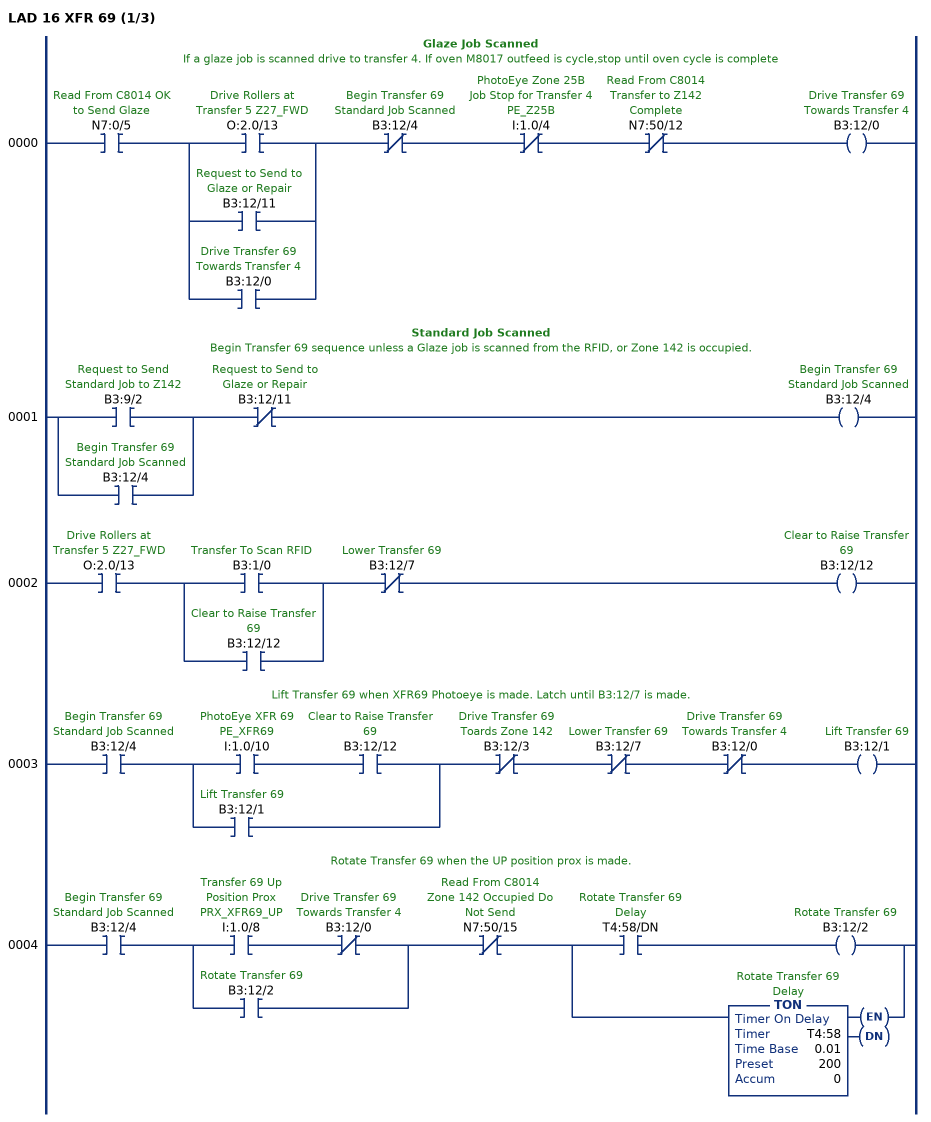
% Rung: 0 %
% TITLE: Glaze Job Scanned %
% If a glaze job is scanned drive to transfer 4. If oven M8017 outfeed is cycle,stop until oven cycle is complete %
SOR XIC N7:0/5 BST XIC O:2.0/13 NXB XIC B3:12/11 NXB XIC B3:12/0 BND XIO B3:12/4 XIO I:1.0/4 XIO N7:50/12 OTE B3:12/0 EOR
%   N7:0/5  "Read From C8014 OK to Send Glaze" %
%   O:2.0/13  Z27_FWD  "Drive Rollers at Transfer 5" %
%   B3:12/11  "Request to Send to Glaze or Repair" %
%   B3:12/0  "Drive Transfer 69 Towards Transfer 4" %
%   B3:12/4  "Begin Transfer 69 Standard Job Scanned" %
%   I:1.0/4  PE_Z25B  "PhotoEye Zone 25B Job Stop for Transfer 4" %
%   N7:50/12  "Read From C8014 Transfer to Z142 Complete" %
% Rung: 1 %
% TITLE: Standard Job Scanned %
% Begin Transfer 69 sequence unless a Glaze job is scanned from the RFID, or Zone 142 is occupied. %
SOR BST XIC B3:9/2 NXB XIC B3:12/4 BND XIO B3:12/11 OTE B3:12/4 EOR
%   B3:9/2  "Request to Send Standard Job to Z142" %
%   B3:12/4  "Begin Transfer 69 Standard Job Scanned" %
%   B3:12/11  "Request to Send to Glaze or Repair" %
% Rung: 2 %
SOR XIC O:2.0/13 BST XIC B3:1/0 NXB XIC B3:12/12 BND XIO B3:12/7 OTE B3:12/12 EOR
%   O:2.0/13  Z27_FWD  "Drive Rollers at Transfer 5" %
%   B3:1/0  "Transfer To Scan RFID" %
%   B3:12/12  "Clear to Raise Transfer 69" %
%   B3:12/7  "Lower Transfer 69" %
% Rung: 3 %
% Lift Transfer 69 when XFR69 Photoeye is made. Latch until B3:12/7 is made. %
SOR XIC B3:12/4 BST XIC I:1.0/10 XIC B3:12/12 NXB XIC B3:12/1 BND XIO B3:12/3 XIO B3:12/7 XIO B3:12/0 OTE B3:12/1 EOR
%   B3:12/4  "Begin Transfer 69 Standard Job Scanned" %
%   I:1.0/10  PE_XFR69  "PhotoEye XFR 69" %
%   B3:12/12  "Clear to Raise Transfer 69" %
%   B3:12/1  "Lift Transfer 69" %
%   B3:12/3  "Drive Transfer 69 Toards Zone 142" %
%   B3:12/7  "Lower Transfer 69" %
%   B3:12/0  "Drive Transfer 69 Towards Transfer 4" %
% Rung: 4 %
% Rotate Transfer 69 when the UP position prox is made. %
SOR XIC B3:12/4 BST XIC I:1.0/8 XIO B3:12/0 NXB XIC B3:12/2 BND XIO N7:50/15 BST XIC T4:58/DN OTE B3:12/2 NXB TON T4:58 0.01 200 0 BND EOR
%   B3:12/4  "Begin Transfer 69 Standard Job Scanned" %
%   I:1.0/8  PRX_XFR69_UP  "Transfer 69 Up Position Prox" %
%   B3:12/0  "Drive Transfer 69 Towards Transfer 4" %
%   B3:12/2  "Rotate Transfer 69" %
%   N7:50/15  "Read From C8014 Zone 142 Occupied Do Not Send" %
%   T4:58  "Rotate Transfer 69 Delay" %

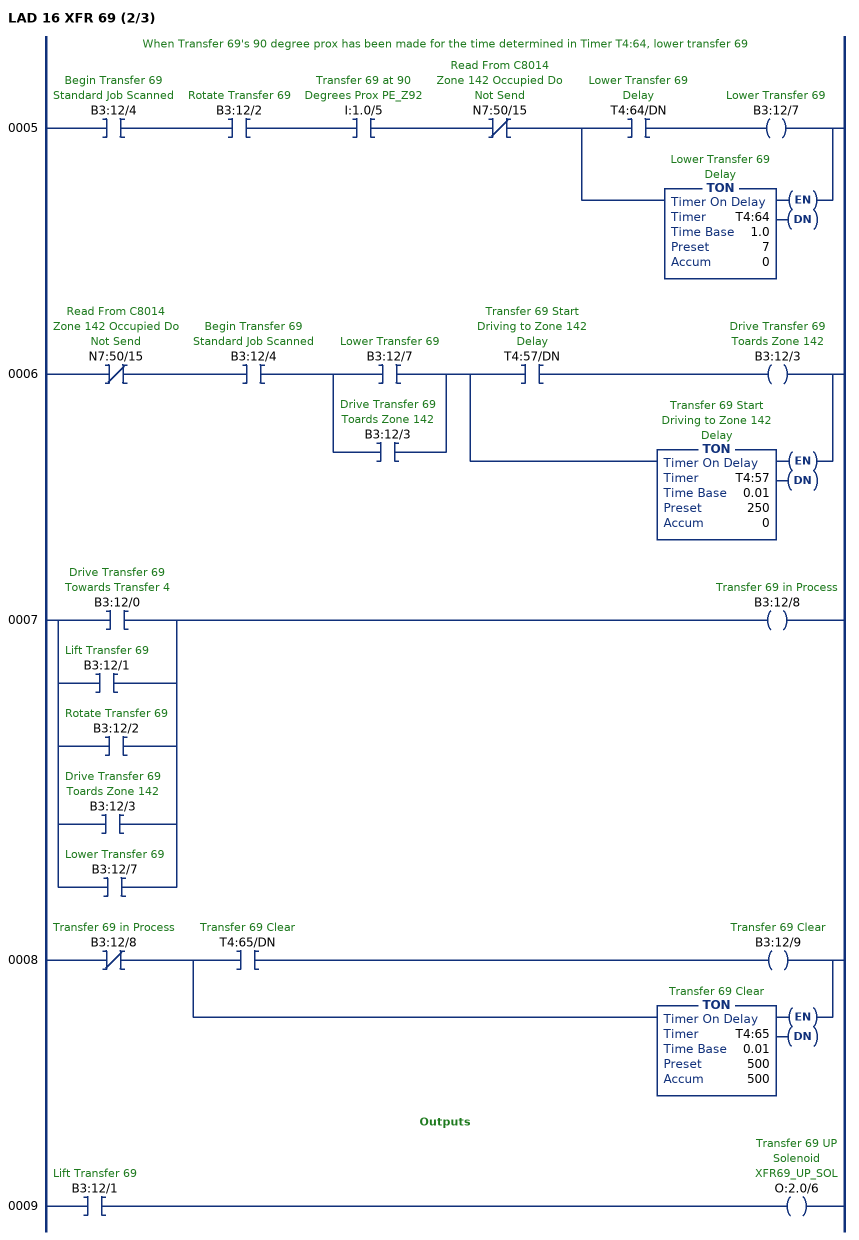
% Rung: 5 %
% When Transfer 69's 90 degree prox has been made for the time determined in Timer T4:64, lower transfer 69 %
SOR XIC B3:12/4 XIC B3:12/2 XIC I:1.0/5 XIO N7:50/15 BST XIC T4:64/DN OTE B3:12/7 NXB TON T4:64 1.0 7 0 BND EOR
%   B3:12/4  "Begin Transfer 69 Standard Job Scanned" %
%   B3:12/2  "Rotate Transfer 69" %
%   I:1.0/5  PE_Z92  "Transfer 69 at 90 Degrees Prox" %
%   N7:50/15  "Read From C8014 Zone 142 Occupied Do Not Send" %
%   T4:64  "Lower Transfer 69 Delay" %
%   B3:12/7  "Lower Transfer 69" %
% Rung: 6 %
SOR XIO N7:50/15 XIC B3:12/4 BST XIC B3:12/7 NXB XIC B3:12/3 BND BST XIC T4:57/DN OTE B3:12/3 NXB TON T4:57 0.01 250 0 BND EOR
%   N7:50/15  "Read From C8014 Zone 142 Occupied Do Not Send" %
%   B3:12/4  "Begin Transfer 69 Standard Job Scanned" %
%   B3:12/7  "Lower Transfer 69" %
%   B3:12/3  "Drive Transfer 69 Toards Zone 142" %
%   T4:57  "Transfer 69 Start Driving to Zone 142 Delay" %
% Rung: 7 %
SOR BST XIC B3:12/0 NXB XIC B3:12/1 NXB XIC B3:12/2 NXB XIC B3:12/3 NXB XIC B3:12/7 BND OTE B3:12/8 EOR
%   B3:12/0  "Drive Transfer 69 Towards Transfer 4" %
%   B3:12/1  "Lift Transfer 69" %
%   B3:12/2  "Rotate Transfer 69" %
%   B3:12/3  "Drive Transfer 69 Toards Zone 142" %
%   B3:12/7  "Lower Transfer 69" %
%   B3:12/8  "Transfer 69 in Process" %
% Rung: 8 %
SOR XIO B3:12/8 BST XIC T4:65/DN OTE B3:12/9 NXB TON T4:65 0.01 500 500 BND EOR
%   B3:12/8  "Transfer 69 in Process" %
%   T4:65  "Transfer 69 Clear" %
%   B3:12/9  "Transfer 69 Clear" %
% Rung: 9 %
% TITLE: Outputs %
SOR XIC B3:12/1 OTE O:2.0/6 EOR
%   B3:12/1  "Lift Transfer 69" %
%   O:2.0/6  XFR69_UP_SOL  "Transfer 69 UP Solenoid" %

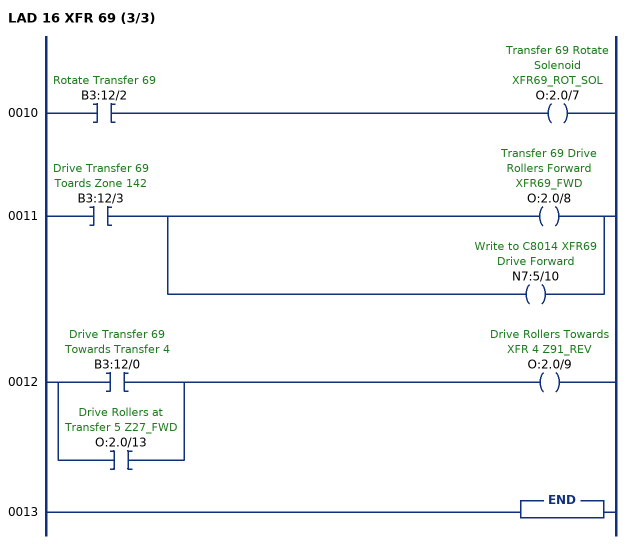
% Rung: 10 %
SOR XIC B3:12/2 OTE O:2.0/7 EOR
%   B3:12/2  "Rotate Transfer 69" %
%   O:2.0/7  XFR69_ROT_SOL  "Transfer 69 Rotate Solenoid" %
% Rung: 11 %
SOR XIC B3:12/3 BST OTE O:2.0/8 NXB OTE N7:5/10 BND EOR
%   B3:12/3  "Drive Transfer 69 Toards Zone 142" %
%   O:2.0/8  XFR69_FWD  "Transfer 69 Drive Rollers Forward" %
%   N7:5/10  "Write to C8014 XFR69 Drive Forward" %
% Rung: 12 %
SOR BST XIC B3:12/0 NXB XIC O:2.0/13 BND OTE O:2.0/9 EOR
%   B3:12/0  "Drive Transfer 69 Towards Transfer 4" %
%   O:2.0/13  Z27_FWD  "Drive Rollers at Transfer 5" %
%   O:2.0/9  Z91_REV  "Drive Rollers Towards XFR 4" %
% Rung: 13 %
SOR END EOR

OTHER DOCUMENTED ADDRESSES
  B3:4/9  "TRANSFER TO TOPCOAT MADE IT PAST THE XFR4"
  B3:4/10  "TRANSFER TO TOPCOAT MADE IT TO PE Z90B OR OVEN"
  B3:5/4  "Latch Zones 26 and 27"
  B3:9/1  "Request to Send to Glaze Sent to C8014"
  B3:9/5  "Transfer to Glazing Area Complete"
  B3:9/6  "Clear to Send to Glazing Area"
  B3:12/5  "Job Scanned Clear Data"
  B3:12/6  "OK to begin Transfer to Z142"
  B3:12/10  "Drive Rollers Towards Zone 142"
  B3:12/15  "Job Scanned Direction Determined Erase RFID Data"
  B3:13/5  "Clear RFID Data One Shot"
  B3:13/6  "Clear RFID Data One Shot"
  I:0.0/8  PR_XFR5_UP
  I:1.0/0  PE_SG21
  I:1.0/6  PRX_XFR69_90  "Transfer 69, 90 Degree Position"
  I:1.0/7  PE_Z90B
  I:1.0/9  PE_Z26
  I:1.0/12  PE_Z34A
  I:3.0/12  PE_Z55B
  I:7.0/11  PR_XFR10_UP
  N7:0/1  "ENTRY TO TOPCOAT B IS FULL"
  N7:1/7  "Write to C8014 Standard Job Scanned From RFID"
  N7:1/8  "Temporary Bit Write to C8014 Sanding Barn To Top Coat B"
  N7:3/5  "From C8011 Request to Send Glaze Job"
  N7:4/2  "DOOR OPEN AT TOP COAT B"
  N7:5/7  "Temporary Bit Jobs From Barn to TCB"
  N7:5/8  "Temporary Bit Write to C8014 Sanding Barn To Top Coat B"
  N7:50/7  "Temporary Bit Write to C8014 Sanding Barn To Top Coat B"
  N7:50/8  "Temporary Bit Write to C8014 Sanding Barn To Top Coat B"
  N7:50/10  "Read From C8014 Transfer to Glaze In Process"
  O:0.0/0  MCR_LED
  O:2.0/11  Z90_REV  "Zone 90 Reverse"
  PE_XFR6_UP  
  PE_Z25_B  
  PE_Z59  
  PE_Z89B  
  PR_XFR8_DH  
  PR_XFR_90  
  PR_XFR_DN  
  PR_XFR_HM  
  ST11:0  ST13  "Extract Material Number"
  ST11:0.0  "RFID Data"
  ST13:1.0  "MAterial Number Present"
  T4:15  "Clear to Cycle M8017 Outfeed"
  T4:59  "Standard Job Scanned Delay. Gives Processor Time to Scan Glaze Material Numbers"
  XFR_6_FWD  

COMMENTS NOT ATTACHED TO A CURRENT RUNG
  T4:31: RAISE TO DRIVE HEIGHT AND RUN XFR4 FWD WAIT FOR PE Z25B
  T4:16: OVEN TO SANDING BARN LOGIC

DATA TABLE (non-zero values as saved)
DATA B3
% B3:0 % 0X0D34 0X2000 0X8856 0XC010 0X0908 0X4088 0X0026 0X0040 0X0000 0X0004
% B3:10 % 0X0000 0X0000 0X0210 0X0040 0X0000 0X0000 0X0000 0X0000 0X0000 0X0000
DATA T4
% .PRE .ACC %
% T4:0 % 25 0
% T4:1 % 50 0
% T4:2 % 50 50
% T4:3 % 100 100
% T4:4 % 1 0
% T4:5 % 200 200
% T4:6 % 400 400
% T4:7 % 50 2
% T4:8 % 1000 0
% T4:9 % 25 25
% T4:10 % 500 0
% T4:11 % 40 0
% T4:12 % 600 600
% T4:13 % 325 0
% T4:14 % 200 200
% T4:15 % 100 0
% T4:16 % 300 0
% T4:17 % 900 0
% T4:18 % 600 0
% T4:19 % 1000 1000
% T4:20 % 100 0
% T4:21 % 100 0
% T4:22 % 40 0
% T4:23 % 10 0
% T4:24 % 100 0
% T4:25 % 500 0
% T4:26 % 50 0
% T4:27 % 50 0
% T4:28 % 10 0
% T4:29 % 10 0
% T4:30 % 10 0
% T4:31 % 1 0
% T4:32 % 100 0
% T4:33 % 100 0
% T4:34 % 1100 0
% T4:35 % 100 0
% T4:36 % 100 0
% T4:37 % 1 0
% T4:38 % 400 0
% T4:39 % 1000 0
% T4:40 % 10 0
% T4:41 % 100 0
% T4:42 % 10 0
% T4:43 % 100 0
% T4:44 % 100 0
% T4:45 % 400 0
% T4:46 % 100 0
% T4:47 % 100 0
% T4:48 % 400 0
% T4:49 % 10 0
% T4:50 % 10 0
% T4:51 % 400 0
% T4:52 % 1000 0
% T4:53 % 500 0
% T4:54 % 200 0
% T4:55 % 5 0
% T4:56 % 50 50
% T4:57 % 250 0
% T4:58 % 200 0
% T4:59 % 50 20
% T4:60 % 2 2
% T4:61 % 100 0
% T4:62 % 200 200
% T4:63 % 200 0
% T4:64 % 7 0
% T4:65 % 500 500
% T4:66 % 25 0
% T4:68 % 100 0
DATA C5
% .PRE .ACC %
% C5:0 % 2 1
% C5:1 % 5 0
% C5:10 % 1000 286
DATA R6
% .LEN .POS %
% R6:1 % 5 4
% R6:2 % 5 4
% R6:3 % 5 4
DATA N7
% N7:0 % 1 256 0 4 0 -32256 0 14 14 0
% N7:10 % 10 10 10 10 10 10 0 0 0 0
% N7:20 % 14 14 14 14 0 0 0 0 0 0
% N7:30 % 21 36 40 43 0 0 0 0 0 0
% N7:40 % 4 38 58 42 0 0 0 0 0 0
% N7:50 % 8 0 17 0 0 0 0 0 0 0
% N7:60 % 3 0 0 0 0 0 0 0 0 0
DATA ST12
% ST12:0 % "71006856"
% ST12:1 % "71085844"
% ST12:2 % "71006856"
% ST12:3 % "71085830"
% ST12:4 % "71085828"
% ST12:5 % "71085845"
% ST12:6 % "71086433"
% ST12:7 % "71086039"
% ST12:8 % "71086002"
% ST12:9 % "71085720"
% ST12:10 % "71086401"
% ST12:11 % "71086393"
% ST12:12 % "71086046"
% ST12:13 % "71085784"
% ST12:14 % "71085800"
% ST12:15 % "71085766"
% ST12:16 % "71086418"
% ST12:17 % "71086035"
% ST12:18 % "71085765"
% ST12:19 % "71085768"
% ST12:20 % "!71006671"
% ST12:21 % "!71006672"
% ST12:22 % "!71064949"
% ST12:23 % "41063579"
% ST12:24 % "41063578"
% ST12:25 % "41063567"
% ST12:26 % "41063568"
% ST12:27 % "41063569"
% ST12:28 % "41063570"
% ST12:29 % "41063571"
% ST12:30 % "41063572"
% ST12:31 % "41063589"
% ST12:32 % "41063590"
% ST12:33 % "41063591"
% ST12:34 % "41063592"
% ST12:35 % "41063593"
% ST12:36 % "41063594"
% ST12:37 % "41063595"
% ST12:38 % "41063596"
% ST12:39 % "41063597"
% ST12:40 % "41063598"
% ST12:41 % "41063599"
% ST12:42 % "41063600"
% ST12:43 % "71086000"
% ST12:44 % "71085788"
% ST12:45 % "71085849"
% ST12:46 % "41063580"
% ST12:47 % "71086383"
% ST12:48 % "spare"
% ST12:49 % "spare"
